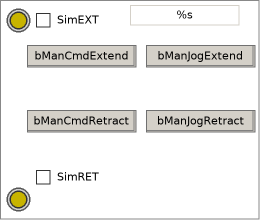
VISUALIZATION VISU_Piston  // 260x220
VAR_IN_OUT
	piston : ST_HmiPiston;
END_VAR
    Label (18,7 95x20)
    Textfield (130,5 109x20), "%s", text variable: piston.Name
    Button (146,45 109x22), "bManJogExtend"
        tap piston.bManJogExtend
    Button (146,110 109x22), "bManJogRetract"
        tap piston.bManJogRetract
    Button (27,110 109x22), "bManCmdRetract"
        tap piston.bManCmdRetract
    Button (27,45 109x22), "bManCmdExtend"
        tap piston.bManCmdExtend
    Checkbox (34,5 84x30), "SimEXT", variable: piston.bSimulateExtended
    Checkbox (34,162 84x30), "SimRET", variable: piston.bSimulateRetracted
    Lamp1 (4,7 29x27), variable: piston.bIsExtendedpiston.bIsExtended, style: Lamp-Lamp1-Yellow
    Lamp1 (4,186 29x27), variable: piston.bIsRetracted, style: Lamp-Lamp1-Yellow
END_VISUALIZATION

(* stored: Version 1.1.0.1, ProductVersion 3.1.4026.18
   Visu VISU_Piston: Id {7f451fe8-3de6-4073-bbb7-7fe519c64520} *)
